(* convert value from 64-bit T_ULARGE_INTEGER to 64-bit T_FILETIME *)
FUNCTION F_FILE_ULargeToFileTime : T_FILETIME
VAR_INPUT
	nULarge		: T_ULARGE_INTEGER;
END_VAR
VAR
END_VAR
(*
-------------------------------------------------------------------------------------------------
Date		Version	Author	Comments
-------------------------------------------------------------------------------------------------
03/08/2012	1.39.00	PB		Initial release

-------------------------------------------------------------------------------------------------
*)

MEMMOVE(ADR(F_FILE_ULargeToFileTime), ADR(nULarge), SIZEOF(nULarge));

END_FUNCTION

(* stored: Version 1.1.0.1, ProductVersion 3.1.4024.15
   POU F_FILE_ULargeToFileTime: Id {789b1e71-d643-4580-a5e2-b17ba3dd9060}, SpecialFunc None *)
